RoboDK station: 3D_Part_V4.rdk

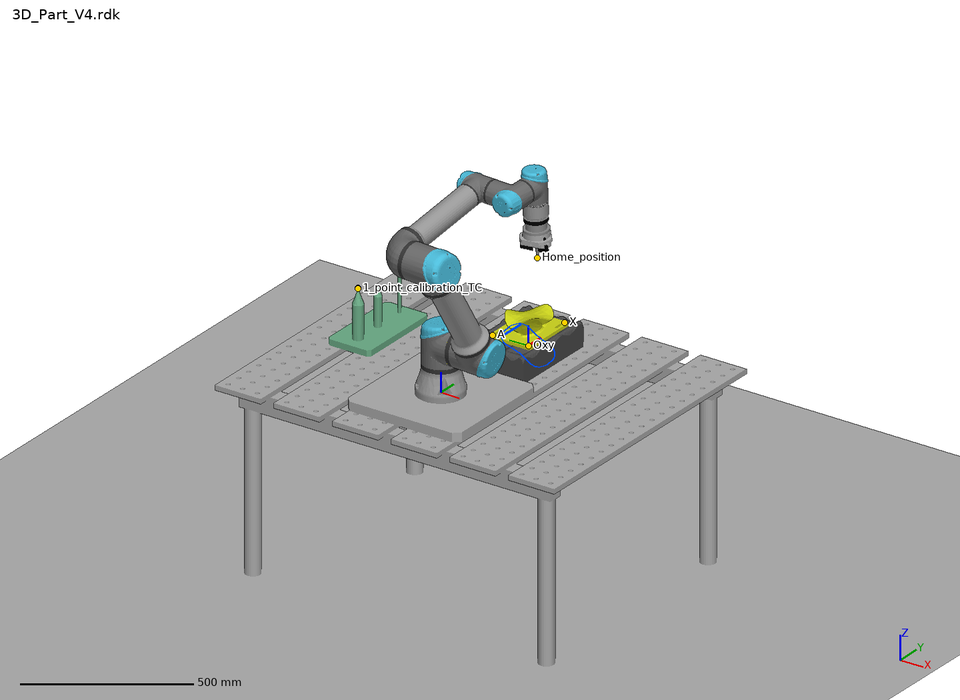
[picture v0: the station drawn from its stored meshes, robots at their saved joint values, targets as dots, program paths as lines]
Station 3D_Part_V4 (saved by RoboDK 5.6.0). Poses are relative to the parent item; angles as X-Y-Z fixed-axis rotations.
  - frame UR5e Base at (0, 0, 30) mm
    - target Home_position (joint target) at (151.97, 268.81, 366.78) mm, rotated rx 178.79 ry -2.3 rz 101.4 deg; joints [86.58, -59.04, -110.78, -97.65, 89.42, -104.81] of UR5e
    - robot UR5e: 6 axes, payload 5 kg, reach 850 mm, repeatability 0.03 mm, weight 18.4 kg
        modified DH rows (alpha deg, a mm, theta deg, d mm): 0, 0, 0, 162.5; 90, 0, 180, 0; 0, 425, 0, 0; 0, 392.25, 0, 133.3; -90, 0, 0, 99.7; 90, 0, 180, 99.6
        joint limits [-360, -360, -360, -360, -360, -360] to [360, 360, 360, 360, 360, 360]; home [0, -90, -90, 0, 90, 0]; saved at [86.58, -59.04, -110.78, -97.65, 89.42, -104.81]
      - tool Gripper, TCP at (0.02, 0, 134.54) mm, size 93 x 134.6 x 99.8 mm, geometry from UR5e
    - target 1_point_calibration_TCP (joint target) at (-409.67, 169.42, 149.93) mm, rotated rx 177.6 ry 0.93 rz 178.1 deg; joints [-38.601, -91.517, 122.976, -122.144, -92.477, -126.732] of UR5e
    - target 2_point_calibration_TCP (joint target) at (-410.25, 171.04, 150.5) mm, rotated rx 176.95 ry 38.31 rz 176.24 deg; joints [-30.106, -71.878, 98.621, -82.617, -108.81, -111.587] of UR5e
    - target 3_point_calibration_TCP (joint target) at (-409.99, 169.96, 150.21) mm, rotated rx 126.21 ry 38.31 rz 176.24 deg; joints [196.668, -105.719, -110.682, -107.023, 51.076, -69.389] of UR5e
    - target 4_point_calibration_TCP (joint target) at (-409.84, 170.1, 150.12) mm, rotated rx 173.91 ry -42.23 rz -175.16 deg; joints [-58.81, -99.027, 150.427, -169.407, -56.512, -142.715] of UR5e
    - target Oxy (Cartesian target) at (100.53, 296.6, 59.24) mm, rotated rx 180 ry 0.32 rz -157.85 deg; joints [96.72, -78.28, -148.41, -43.22, 89.69, -195.43] of UR5e
    - target X (Cartesian target) at (99.52, 481.53, 59.5) mm, rotated rx 179.89 ry 0.3 rz 180 deg; joints [94.201, -103.645, -122.326, -43.943, 89.694, -175.799] of UR5e
    - target A (Cartesian target) at (-24.47, 295.97, 58.57) mm, rotated rx 179.68 ry 0.01 rz 113.97 deg; joints [121.68, -75.14, -150.51, -44.4, 89.68, -82.29] of UR5e
  - object Floor at (-40, 90, -610) mm, size 3000 x 3000 x 0 mm, geometry from Floor.stl
  - object Table at (0, 200, 0) mm, size 1193.8 x 965.2 x 609.6 mm, geometry from Stol.stl
  - object Postolje_UR5e at (0, 0, 0) mm, rotated rx 90 ry 0 rz 0 deg, size 400 x 30 x 400 mm, geometry from Postolje_UR5e.STEP
  - object sponge at (29.84, 379.94, 30) mm, rotated rx 90 ry 0 rz 0 deg, size 200 x 50.9 x 301 mm, geometry from sponge.STEP
  - object Calibration_Gauge at (-410, 270, 0) mm, rotated rx 0 ry 0 rz 90 deg, size 300 x 150 x 180 mm, geometry from kalibracijski_siljak_fiksni_3.stl
  - object 3D_Part at (37, 389, 189) mm, rotated rx 0.3 ry 0.11 rz -89.69 deg, size 200 x 145 x 75.1 mm, geometry from 3D_Part_V3.STEP
  - object sponge at (29.5, 380, 0) mm, rotated rx 90 ry 0 rz 0 deg, size 200 x 50.9 x 301 mm, geometry from sponge.STEP
  - frame Frame_Part at (100.25, 296, 89.5) mm, rotated rx 0 ry 0 rz 90 deg
    - object 3D_Curve at (93, 63, 40) mm, rotated rx 0 ry -90 rz 90 deg, geometry from Imported curve
  - machining project Curve settings: rotZ(0) | rotX(0)*rotY(0) | rotz(0) | onStart | onPathStart | onApproach | onPoint | onRetract | onFinish | SetRPM(%1) | SetTool(%1) | Extruder(%1) | default | default | OutOnMov(%1) | OutOffMov(%1) | onPathFinish | M_RunCode(%1)
  - program Curve (79 instructions, listed below)
  - program Main_Program (5 instructions, listed below)
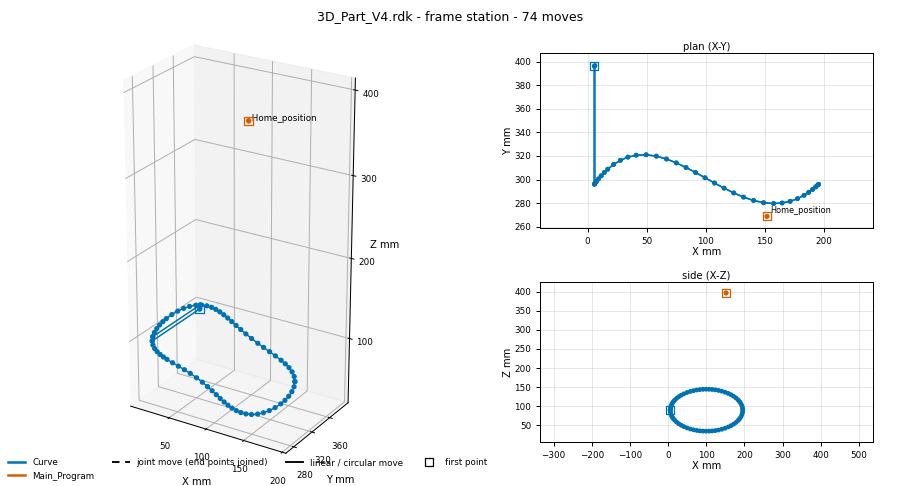
[picture p0: tool path of 3D_Part_V4.rdk in frame station, 74 of 74 moves have a stored position in this frame; points joined in program order, loops and branches not executed]

--- program Curve (robot UR5e) ---
  Smooth(1)
  Set speed (1000.0 mm/s)
  Set Ref.: Frame_Part
  Set Tool: Gripper
  Show Gripper
  MoveJ 1 to (100, 94.5, 0) mm, rotated rx 90 ry 90 rz -90 deg; joints [109.469, -59.624, -134.471, -75.906, 90, -160.531]
  MoveL 2 to (100, 94.5, 0) mm, rotated rx 90 ry 90 rz -90 deg; joints [109.469, -59.624, -134.471, -75.906, 90, -160.531]
  MoveL 3 to (0, 94.5, 0) mm, rotated rx 90 ry 90 rz -90 deg; joints [109.469, -68.399, -146.428, -55.173, 90, -160.531]
  MoveL 4 to (0, 94.5, 0) mm, rotated rx 90 ry 90 rz -90 deg; joints [109.469, -68.399, -146.428, -55.173, 90, -160.531]
  Set speed (50.0 mm/s)
  MoveL 5 to (0.61, 94.06, -5.31) mm, rotated rx 90 ry 90 rz -90 deg; joints [110.516, -68.275, -146.384, -55.341, 90, -159.484]
  MoveL 6 to (2.24, 92.83, -10.29) mm, rotated rx 90 ry 90 rz -90 deg; joints [111.424, -68.214, -146.126, -55.659, 90, -158.576]
  MoveL 7 to (4.53, 91, -14.79) mm, rotated rx 90 ry 90 rz -90 deg; joints [112.176, -68.226, -145.716, -56.057, 90, -157.824]
  MoveL 8 to (7.18, 88.74, -18.87) mm, rotated rx 90 ry 90 rz -90 deg; joints [112.796, -68.315, -145.205, -56.48, 90, -157.204]
  MoveL 9 to (9.97, 86.11, -22.6) mm, rotated rx 90 ry 90 rz -90 deg; joints [113.303, -68.482, -144.629, -56.889, 90, -156.697]
  MoveL 10 to (12.78, 83.16, -26.06) mm, rotated rx 90 ry 90 rz -90 deg; joints [113.721, -68.732, -144.007, -57.261, 90, -156.279]
  MoveL 11 to (16.82, 78.14, -30.86) mm, rotated rx 90 ry 90 rz -90 deg; joints [114.205, -69.277, -143.013, -57.71, 90, -155.795]
  MoveL 12 to (20.32, 72.45, -35.23) mm, rotated rx 90 ry 90 rz -90 deg; joints [114.534, -70.03, -141.992, -57.978, 90, -155.466]
  MoveL 13 to (23.02, 66.05, -39.25) mm, rotated rx 90 ry 90 rz -90 deg; joints [114.728, -71.012, -140.963, -58.025, 90, -155.272]
  MoveL 14 to (24.64, 59.06, -42.85) mm, rotated rx 90 ry 90 rz -90 deg; joints [114.794, -72.212, -139.968, -57.821, 90, -155.206]
  MoveL 15 to (24.99, 50.59, -46.37) mm, rotated rx 90 ry 90 rz -90 deg; joints [114.728, -73.804, -138.913, -57.283, 90, -155.272]
  MoveL 16 to (23.8, 41.94, -49.21) mm, rotated rx 90 ry 90 rz -90 deg; joints [114.542, -75.549, -137.971, -56.479, 90, -155.458]
  MoveL 17 to (21.37, 33.34, -51.39) mm, rotated rx 90 ry 90 rz -90 deg; joints [114.267, -77.373, -137.134, -55.493, 90, -155.733]
  MoveL 18 to (18.07, 24.95, -52.99) mm, rotated rx 90 ry 90 rz -90 deg; joints [113.93, -79.211, -136.379, -54.409, 90, -156.07]
  MoveL 19 to (14.18, 16.76, -54.08) mm, rotated rx 90 ry 90 rz -90 deg; joints [113.548, -81.041, -135.674, -53.285, 90, -156.452]
  MoveL 20 to (9.92, 8.67, -54.74) mm, rotated rx 90 ry 90 rz -90 deg; joints [113.125, -82.859, -134.985, -52.156, 90, -156.875]
  MoveL 21 to (5.47, 0.64, -55) mm, rotated rx 90 ry 90 rz -90 deg; joints [112.666, -84.654, -134.288, -51.058, 90, -157.334]
  MoveL 22 to (1.01, -7.39, -54.86) mm, rotated rx 90 ry 90 rz -90 deg; joints [112.171, -86.416, -133.563, -50.02, 90, -157.829]
  MoveL 23 to (-3.33, -15.46, -54.31) mm, rotated rx 90 ry 90 rz -90 deg; joints [111.638, -88.136, -132.791, -49.073, 90, -158.362]
  MoveL 24 to (-7.36, -23.65, -53.34) mm, rotated rx 90 ry 90 rz -90 deg; joints [111.062, -89.803, -131.953, -48.244, 90, -158.938]
  MoveL 25 to (-10.92, -31.99, -51.89) mm, rotated rx 90 ry 90 rz -90 deg; joints [110.437, -91.398, -131.033, -47.569, 90, -159.563]
  MoveL 26 to (-13.76, -40.48, -49.89) mm, rotated rx 90 ry 90 rz -90 deg; joints [109.757, -92.897, -130.017, -47.086, 90, -160.243]
  MoveL 27 to (-15.64, -48.99, -47.3) mm, rotated rx 90 ry 90 rz -90 deg; joints [109.025, -94.253, -128.91, -46.837, 90, -160.975]
  MoveL 28 to (-16.33, -57.46, -44.02) mm, rotated rx 90 ry 90 rz -90 deg; joints [108.235, -95.44, -127.714, -46.846, 90, -161.765]
  MoveL 29 to (-15.86, -64.67, -40.55) mm, rotated rx 90 ry 90 rz -90 deg; joints [107.501, -96.314, -126.613, -47.073, 90, -162.499]
  MoveL 30 to (-14.43, -71.4, -36.6) mm, rotated rx 90 ry 90 rz -90 deg; joints [106.747, -97.012, -125.51, -47.477, 90, -163.253]
  MoveL 31 to (-12.17, -77.63, -32.1) mm, rotated rx 90 ry 90 rz -90 deg; joints [105.963, -97.558, -124.417, -48.025, 90, -164.037]
  MoveL 32 to (-9.33, -83.18, -27.08) mm, rotated rx 90 ry 90 rz -90 deg; joints [105.158, -97.964, -123.377, -48.659, 90, -164.842]
  MoveL 33 to (-6.86, -87.07, -22.65) mm, rotated rx 90 ry 90 rz -90 deg; joints [104.493, -98.208, -122.604, -49.188, 90, -165.507]
  MoveL 34 to (-4.38, -90.42, -17.74) mm, rotated rx 90 ry 90 rz -90 deg; joints [103.797, -98.396, -121.902, -49.703, 90, -166.203]
  MoveL 35 to (-2.18, -93.08, -12.32) mm, rotated rx 90 ry 90 rz -90 deg; joints [103.068, -98.538, -121.309, -50.152, 90, -166.932]
  MoveL 36 to (-0.59, -94.86, -6.36) mm, rotated rx 90 ry 90 rz -90 deg; joints [102.303, -98.646, -120.878, -50.476, 90, -167.697]
  MoveL 37 to (0, -95.5, 0) mm, rotated rx 90 ry 90 rz -90 deg; joints [101.523, -98.723, -120.672, -50.605, 90, -168.477]
  MoveL 38 to (0, -95.5, 0) mm, rotated rx 90 ry 90 rz -90 deg; joints [101.523, -98.723, -120.672, -50.605, 90, -168.477]
  MoveL 39 to (-0.59, -94.86, 6.36) mm, rotated rx 90 ry 90 rz -90 deg; joints [100.772, -98.769, -120.729, -50.502, 90, -169.228]
  MoveL 40 to (-2.18, -93.08, 12.34) mm, rotated rx 90 ry 90 rz -90 deg; joints [100.09, -98.778, -121.02, -50.203, 90, -169.91]
  MoveL 41 to (-4.4, -90.4, 17.78) mm, rotated rx 90 ry 90 rz -90 deg; joints [99.486, -98.741, -121.486, -49.773, 90, -170.514]
  MoveL 42 to (-6.86, -87.06, 22.66) mm, rotated rx 90 ry 90 rz -90 deg; joints [98.955, -98.652, -122.068, -49.28, 90, -171.045]
  MoveL 43 to (-9.35, -83.15, 27.11) mm, rotated rx 90 ry 90 rz -90 deg; joints [98.479, -98.499, -122.735, -48.766, 90, -171.521]
  MoveL 44 to (-12.19, -77.58, 32.15) mm, rotated rx 90 ry 90 rz -90 deg; joints [97.951, -98.199, -123.653, -48.148, 90, -172.049]
  MoveL 45 to (-14.45, -71.34, 36.65) mm, rotated rx 90 ry 90 rz -90 deg; joints [97.491, -97.755, -124.632, -47.614, 90, -172.509]
  MoveL 46 to (-15.88, -64.51, 40.64) mm, rotated rx 90 ry 90 rz -90 deg; joints [97.091, -97.144, -125.643, -47.212, 90, -172.909]
  MoveL 47 to (-16.33, -57.35, 44.07) mm, rotated rx 90 ry 90 rz -90 deg; joints [96.758, -96.369, -126.642, -46.988, 90, -173.242]
  MoveL 48 to (-15.61, -48.82, 47.35) mm, rotated rx 90 ry 90 rz -90 deg; joints [96.454, -95.279, -127.752, -46.968, 90, -173.546]
  MoveL 49 to (-13.71, -40.27, 49.95) mm, rotated rx 90 ry 90 rz -90 deg; joints [96.231, -94.017, -128.786, -47.197, 90, -173.769]
  MoveL 50 to (-10.86, -31.83, 51.92) mm, rotated rx 90 ry 90 rz -90 deg; joints [96.085, -92.622, -129.734, -47.644, 90, -173.915]
  MoveL 51 to (-7.29, -23.5, 53.36) mm, rotated rx 90 ry 90 rz -90 deg; joints [96.006, -91.119, -130.608, -48.273, 90, -173.994]
  MoveL 52 to (-3.25, -15.32, 54.33) mm, rotated rx 90 ry 90 rz -90 deg; joints [95.991, -89.543, -131.411, -49.046, 90, -174.009]
  MoveL 53 to (1.08, -7.25, 54.86) mm, rotated rx 90 ry 90 rz -90 deg; joints [96.037, -87.909, -132.161, -49.93, 90, -173.963]
  MoveL 54 to (5.54, 0.77, 55) mm, rotated rx 90 ry 90 rz -90 deg; joints [96.145, -86.227, -132.877, -50.897, 90, -173.855]
  MoveL 55 to (9.98, 8.79, 54.74) mm, rotated rx 90 ry 90 rz -90 deg; joints [96.319, -84.506, -133.575, -51.919, 90, -173.681]
  MoveL 56 to (14.25, 16.9, 54.07) mm, rotated rx 90 ry 90 rz -90 deg; joints [96.567, -82.749, -134.279, -52.971, 90, -173.433]
  MoveL 57 to (18.15, 25.14, 52.96) mm, rotated rx 90 ry 90 rz -90 deg; joints [96.901, -80.964, -135.014, -54.021, 90, -173.099]
  MoveL 58 to (21.44, 33.53, 51.35) mm, rotated rx 90 ry 90 rz -90 deg; joints [97.338, -79.167, -135.809, -55.024, 90, -172.662]
  MoveL 59 to (23.83, 42.05, 49.18) mm, rotated rx 90 ry 90 rz -90 deg; joints [97.897, -77.386, -136.691, -55.923, 90, -172.103]
  MoveL 60 to (25, 50.69, 46.33) mm, rotated rx 90 ry 90 rz -90 deg; joints [98.607, -75.64, -137.701, -56.659, 90, -171.393]
  MoveL 61 to (24.64, 59.1, 42.83) mm, rotated rx 90 ry 90 rz -90 deg; joints [99.471, -74.022, -138.834, -57.144, 90, -170.529]
  MoveL 62 to (23.01, 66.1, 39.22) mm, rotated rx 90 ry 90 rz -90 deg; joints [100.357, -72.754, -139.918, -57.328, 90, -169.643]
  MoveL 63 to (20.31, 72.48, 35.22) mm, rotated rx 90 ry 90 rz -90 deg; joints [101.337, -71.674, -141.042, -57.284, 90, -168.663]
  MoveL 64 to (16.78, 78.2, 30.81) mm, rotated rx 90 ry 90 rz -90 deg; joints [102.412, -70.777, -142.18, -57.043, 90, -167.588]
  MoveL 65 to (12.77, 83.18, 26.04) mm, rotated rx 90 ry 90 rz -90 deg; joints [103.569, -70.058, -143.287, -56.655, 90, -166.431]
  MoveL 66 to (9.97, 86.11, 22.6) mm, rotated rx 90 ry 90 rz -90 deg; joints [104.396, -69.663, -143.995, -56.342, 90, -165.604]
  MoveL 67 to (7.17, 88.74, 18.87) mm, rotated rx 90 ry 90 rz -90 deg; joints [105.281, -69.324, -144.671, -56.005, 90, -164.719]
  MoveL 68 to (4.52, 91.01, 14.79) mm, rotated rx 90 ry 90 rz -90 deg; joints [106.235, -69.033, -145.295, -55.673, 90, -163.765]
  MoveL 69 to (2.23, 92.83, 10.28) mm, rotated rx 90 ry 90 rz -90 deg; joints [107.262, -68.784, -145.832, -55.384, 90, -162.738]
  MoveL 70 to (0.61, 94.06, 5.33) mm, rotated rx 90 ry 90 rz -90 deg; joints [108.351, -68.573, -146.23, -55.197, 90, -161.649]
  Set speed (1000.0 mm/s)
  MoveL 71 to (0.61, 94.06, 5.33) mm, rotated rx 90 ry 90 rz -90 deg; joints [108.351, -68.573, -146.23, -55.197, 90, -161.649]
  MoveL 72 to (100.61, 94.06, 5.33) mm, rotated rx 90 ry 90 rz -90 deg; joints [108.351, -59.833, -134.287, -75.88, 90, -161.649]

--- program Main_Program (robot UR5e) ---
  MoveJ (Home_position)
  Set Ref.: UR5e Base
  Set Tool: Gripper
  Call Curve
  MoveJ (Home_position)
